(* CODESYS project Projeto_Prensa.project

Project tree, tasks and I/O mapping:
  Device : CODESYS Control Win V3, 3S - Smart Software Solutions GmbH, order no. 305021, version 3.5.11.30
    application Application
      libraries: Standard, * (System)
      task MainTask (cyclic, interval t#20ms, priority 1) calls PLC_PRG
      task VISU_TASK (cyclic, interval 100 ms, priority 31) calls VisuElems.Visu_Prg
      program PLC_PRG [LD]
      Symbols
      visualisation Visualization
  libraries: VisuSymbols, 3.5.10.0 (System)
  text list GlobalTextList
*)

// Device/Application/PLC_PRG
PROGRAM PLC_PRG
VAR
	I7: BOOL; //B1
	I0: BOOL; //S1
	I1: BOOL; //S2
	I2: BOOL; //S3
	I3: BOOL; //S4
	I4: BOOL; //S5
	I5: BOOL; //S6
	M0: BOOL; //K1
	M1: BOOL; //K2
	M2: BOOL; //K3
	M3: BOOL; //K4
	M4: BOOL; //K5
	M5: BOOL; //B3
	Q0: BOOL; //Y1
	Q1: BOOL; //Y2
	Q2: BOOL; //Y3
	Q3: BOOL; //Y4
	Q4: BOOL; //Y5
	ED0: BYTE;
	AB0: BYTE;
END_VAR
VAR // added by the converter: edge detectors and wires of the graphical bodies
    _w1 : BOOL;
END_VAR

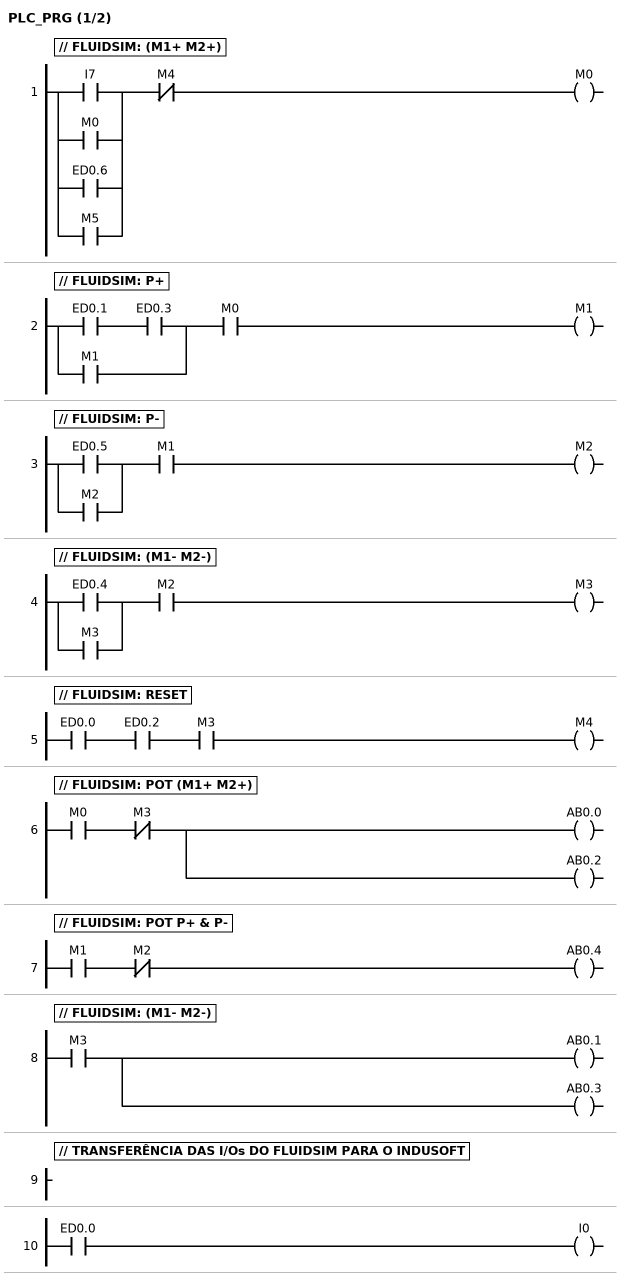
// NETWORK 1
// label: // FLUIDSIM: (M1+ M2+)
M0 := (I7 OR M0 OR ED0.6 OR M5) AND NOT M4;

// NETWORK 2
// label: // FLUIDSIM: P+
M1 := (ED0.1 AND ED0.3 OR M1) AND M0;

// NETWORK 3
// label: // FLUIDSIM: P-
M2 := (ED0.5 OR M2) AND M1;

// NETWORK 4
// label: // FLUIDSIM: (M1- M2-)
M3 := (ED0.4 OR M3) AND M2;

// NETWORK 5
// label: // FLUIDSIM: RESET
M4 := ED0.0 AND ED0.2 AND M3;

// NETWORK 6
// label: // FLUIDSIM: POT (M1+ M2+)
_w1 := M0 AND NOT M3;
AB0.0 := _w1;
AB0.2 := _w1;

// NETWORK 7
// label: // FLUIDSIM: POT P+ & P-
AB0.4 := M1 AND NOT M2;

// NETWORK 8
// label: // FLUIDSIM: (M1- M2-)
AB0.1 := M3;
AB0.3 := M3;

// NETWORK 9
// label: // TRANSFERÊNCIA DAS I/Os DO FLUIDSIM PARA O INDUSOFT

// NETWORK 10
I0 := ED0.0;

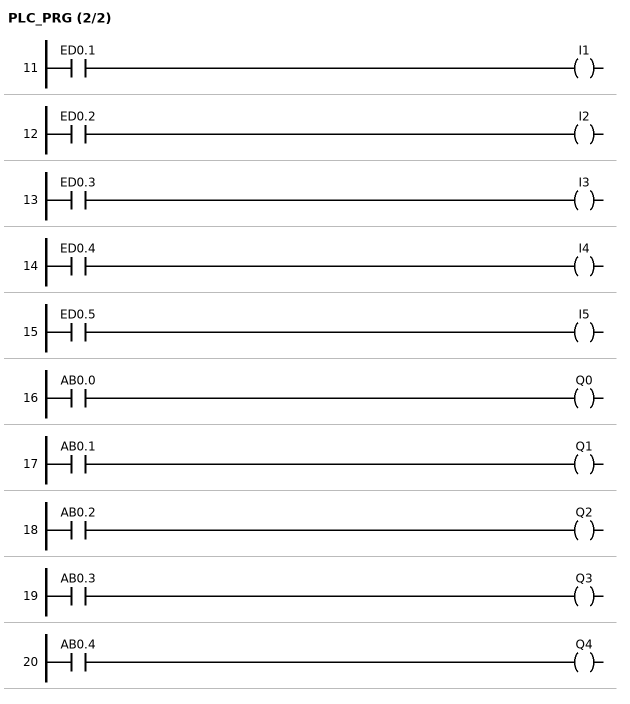
// NETWORK 11
I1 := ED0.1;

// NETWORK 12
I2 := ED0.2;

// NETWORK 13
I3 := ED0.3;

// NETWORK 14
I4 := ED0.4;

// NETWORK 15
I5 := ED0.5;

// NETWORK 16
Q0 := AB0.0;

// NETWORK 17
Q1 := AB0.1;

// NETWORK 18
Q2 := AB0.2;

// NETWORK 19
Q3 := AB0.3;

// NETWORK 20
Q4 := AB0.4;

END_PROGRAM

// Device/Application/Visualization
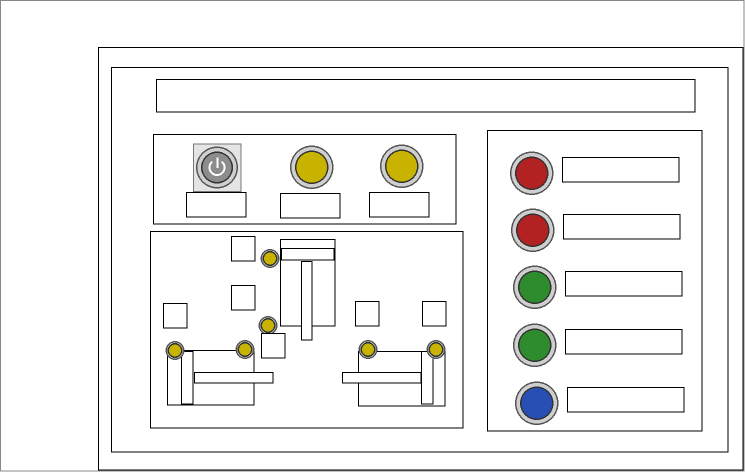
VISUALIZATION Visualization  // 745x472
    Rectangle (98,47 645x423)
    RoundedRectangle (111,67 617x385)
    Lamp1 (692,296 2x0), style: Lamp-Lamp1-Yellow
    RoundedRectangle (150,231 313x197)
    Group (280,239 55x101)
        Rectangle (0,0 55x87)
        Rectangle (21,22 11x79)
        Rectangle (1,9 53x12)
    Rectangle (183,335 55x87), angle 270
    Rectangle (161,372 53x12), angle 270
    Rectangle (228,339 11x79), angle 270
    Rectangle (374,336 55x87), angle 270
    Rectangle (401,372 53x12), angle 270
    Rectangle (376,339 11x79), angle 270
    Lamp1 (425,329 22x41), variable: PLC_PRG.I2, style: Lamp-Lamp1-Yellow
    Lamp1 (357,329 22x41), variable: PLC_PRG.I3, style: Lamp-Lamp1-Yellow
    Lamp1 (257,305 22x41), variable: PLC_PRG.I5, style: Lamp-Lamp1-Yellow
    Lamp1 (259,238 22x41), variable: PLC_PRG.I4, style: Lamp-Lamp1-Yellow
    Lamp1 (164,330 22x41), variable: PLC_PRG.I0, style: Lamp-Lamp1-Yellow
    Lamp1 (234,329 22x41), variable: PLC_PRG.I1, style: Lamp-Lamp1-Yellow
    RoundedRectangle (487,130 215x301)
    Lamp1 (505,148 53x50), variable: PLC_PRG.Q0, style: Lamp-Lamp1-Red
    Rectangle (562,157 117x25), "Solenóide Y1"
    Lamp1 (506,205 53x50), variable: PLC_PRG.Q1, style: Lamp-Lamp1-Red
    Rectangle (563,214 117x25), "Solenóide Y2"
    Lamp1 (508,262 53x50), variable: PLC_PRG.Q2, style: Lamp-Lamp1-Green
    Rectangle (565,271 117x25), "Solenóide Y3"
    Lamp1 (508,320 53x50), variable: PLC_PRG.Q3, style: Lamp-Lamp1-Green
    Rectangle (565,329 117x25), "Solenóide Y4"
    Lamp1 (510,378 53x50), variable: PLC_PRG.Q4, style: Lamp-Lamp1-Blue
    Rectangle (567,387 117x25), "Solenóide Y5"
    RoundedRectangle (153,134 303x90)
    PowerSwitch (193,142 48x51), variable: PLC_PRG.M5, behaviour: TOGGLE, style: Switch-PowerSwitch-Gray
    Rectangle (186,192 60x25), "Botão B3"
    Lamp1 (285,142 53x50), variable: PLC_PRG.ED0.6, style: Lamp-Lamp1-Yellow
    Lamp1 (375,141 53x50), variable: PLC_PRG.I7, style: Lamp-Lamp1-Yellow
    Rectangle (280,193 60x25), "Botão B2"
    Rectangle (369,192 60x25), "Botão B1"
    Rectangle (231,236 24x25), "S5"
    Rectangle (231,285 24x25), "S6"
    Rectangle (163,303 24x25), "S1"
    Rectangle (261,333 24x25), "S2"
    Rectangle (355,301 24x25), "S4"
    Rectangle (422,301 24x25), "S3"
    RoundedRectangle (156,79 539x33), "CONTROLE E MONITORAMENTO - PRENSA ELETROPNEUMÁTICA"
END_VISUALIZATION
